// TIA Portal V17 export
// export: Created 2023-04-20T08:24:45.6440987Z, ExportSetting WithDefaults, DisplayName Totally Integrated Automation Portal, DisplayVersion V17, DisplayName TIA Portal Openness, DisplayVersion V17, DisplayName TIA Portal Version Control Interface, DisplayVersion V17, DisplayName STEP 7 Professional, DisplayVersion V17, DisplayName STEP 7 Safety, DisplayVersion V17, DisplayName WinCC Advanced, DisplayVersion V17
FUNCTION "NormScalev2" : Void   // FC1, LAD
{ S7_Optimized_Access := 'TRUE' }
VERSION : 0.1
// stored: AutoNumber true, IsIECCheckEnabled false, SetENOAutomatically false, UDAEnableTagReadback false
   VAR_INPUT
      Analog_Input : UInt;
   END_VAR
   VAR_OUTPUT
      Analog_value : Real;
   END_VAR
   VAR_TEMP
      norm_analog_input : Real;
   END_VAR
   VAR CONSTANT
      Upper_int : UInt := 27648;
      Lower_int : UInt := 0;
      Upper_Real : Real := 100.0;
      Lower_Real : Real := 0.0;
   END_VAR
BEGIN

REGION Network 1
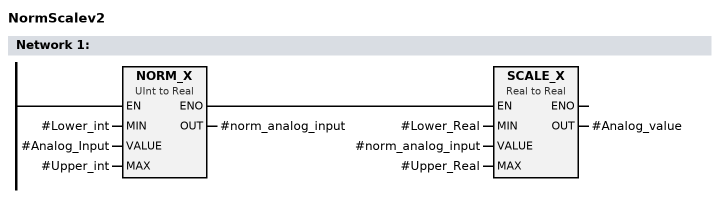
   RUNG wire#powerrail
      { S7_Templates := "[SrcType := UInt, DestType := Real]" } Normalize(min := #Lower_int, value := #Analog_Input, max := #Upper_int, out => #norm_analog_input)
      { S7_Templates := "[SrcType := Real, DestType := Real]" } Scale(min := #Lower_Real, value := #norm_analog_input, max := #Upper_Real, out => #Analog_value)
   END_RUNG
   // the same network as SCL:
   #norm_analog_input := NORM_X(MIN := #Lower_int, VALUE := #Analog_Input, MAX := #Upper_int);
   #Analog_value := SCALE_X(MIN := #Lower_Real, VALUE := #norm_analog_input, MAX := #Upper_Real);
END_REGION
END_FUNCTION
